METHOD PRIVATE T13_TestPowerForTopElement
VAR_INST
	iStep: INT;
END_VAR
IF (TcUnit.TEST_ORDERED ('T13_TestPowerForTopElement')) THEN
	GVL_Variable.fbPB1.ExecuteEveryCycle_Test ();
	GVL_Variable.fbPB1.ExecuteEveryCycle_Operation ();
	GVL_Variable.fbPB1.ExecuteEveryCycle_Status ();
	 CASE iStep	OF
	0	:
		GVL.fbSS1.SetFlag (bState	:= FALSE);
		GVL.fbSTO.SetFlag (bState	:= FALSE);
		AssertFalse		(Condition := GVL.fbSS1.GetFlag (), Message := 'K0 - T01 - bledny stan SS1');
		AssertFalse		(Condition := GVL.fbSTO.GetFlag (), Message := 'K0 - T02 - bledny stan SSO');
		GVL_Variable.fbPB1.PowerTurnOn ();
		iStep			:= iStep + 10;
	10	:
		AssertFalse (Condition := GVL_Variable.fbPB1.stEvents.arrState [1], 				Message := 'T10 - 01 - bledny stan bledu SS1');
		AssertFalse (Condition := GVL_Variable.fbPB1.stEvents.arrState [2], 				Message := 'T10 - 02 - bledny stan bledu STO');
		AssertTrue (Condition := GVL_Variable.fbPB1.stPower.cmdTurnOn.IsBusy (), 			Message := 'T10 - 03 - bledny stan trwa');
		AssertTrue (Condition := GVL_Variable.fbPB1.stPower.cmdTurnOn.IsFirstCycle (), 	Message := 'T10 - 05 - bledny pierwszy cykl');
		AssertFalse (Condition := GVL_Variable.fbPB1.stPower.cmdTurnOn.IsLastCycle (), 	Message := 'T10 - 06 - bledny ostatni cykl');
		AssertFalse (Condition := GVL_Variable.fbPB1.PowerGetStatus (), 					Message := 'T10 - 04 - bledny status');
		iStep			:= iStep + 10;
	20	:
		AssertTrue (Condition := GVL_Variable.fbPB1.stEvents.arrState [1], 					Message := 'T20 - 01 - bledny stan bledu SS1');
		AssertTrue (Condition := GVL_Variable.fbPB1.stEvents.arrState [2], 					Message := 'T20 - 02 - bledny stan bledu STO');
		AssertFalse (Condition := GVL_Variable.fbPB1.stPower.cmdTurnOn.IsBusy (), 			Message := 'T20 - 03 - bledny stan trwa');
		AssertFalse (Condition := GVL_Variable.fbPB1.stPower.cmdTurnOn.IsFirstCycle (),	Message := 'T20 - 05 - bledny pierwszy cykl');
		AssertFalse (Condition := GVL_Variable.fbPB1.stPower.cmdTurnOn.IsLastCycle (),	 	Message := 'T20 - 06 - bledny ostatni cykl');
		AssertFalse (Condition := GVL_Variable.fbPB1.PowerGetStatus (), 					Message := 'T20 - 04 - bledny status');
		GVL.fbSS1.SetFlag (bState	:= TRUE);
		GVL.fbSTO.SetFlag (bState	:= TRUE);
		iStep			:= iStep + 10;
	30	:
		iStep			:= iStep + 10;
	40	:
		GVL_Variable.fbPB1.PowerTurnOn ();
		iStep 			:= iStep + 10;
	50	:
		AssertTrue (Condition := GVL_Variable.fbPB1.stEvents.arrState [1], 				Message := 'T50 - 01 - bledny stan bledu SS1');
		AssertTrue (Condition := GVL_Variable.fbPB1.stEvents.arrState [2], 				Message := 'T50 - 02 - bledny stan bledu STO');
		AssertTrue (Condition := GVL_Variable.fbPB1.stPower.cmdTurnOn.IsBusy (), 		Message := 'T50 - 03 - bledny stan trwa');
		AssertFalse (Condition := GVL_Variable.fbPB1.PowerGetStatus (), 					Message := 'T50 - 04 - bledny status');
		iStep			:= iStep + 10;
	60	:
		AssertFalse (Condition := GVL_Variable.fbPB1.stEvents.arrState [1], 			Message := 'T60 - 01 - bledny stan bledu SS1');
		AssertFalse (Condition := GVL_Variable.fbPB1.stEvents.arrState [2], 			Message := 'T60 - 02 - bledny stan bledu STO');
		AssertTrue (Condition := GVL_Variable.fbPB1.stPower.cmdTurnOn.IsBusy (), 		Message := 'T60 - 03 - bledny stan trwa');
		AssertFalse (Condition := GVL_Variable.fbPB1.PowerGetStatus (), 					Message := 'T60 - 04 - bledny status');
		iStep			:= iStep + 10;
	70	:
		AssertTrue (Condition := GVL_Variable.fbPB1.stPower.cmdTurnOn.IsBusy (), 		Message := 'T70 - 03 - bledny stan trwa');
		AssertFalse (Condition := GVL_Variable.fbPB1.PowerGetStatus (), 					Message := 'T70 - 04 - bledny status');
		iStep			:= iStep + 10;
	80	:
		AssertTrue (Condition := GVL_Variable.fbPB1.stPower.cmdTurnOn.IsBusy (), 		Message := 'T80 - 03 - bledny stan trwa');
		AssertFalse (Condition := GVL_Variable.fbPB1.PowerGetStatus (), 					Message := 'T80 - 04 - bledny status');
		iStep			:= iStep + 10;
	90	:
		AssertTrue (Condition := GVL_Variable.fbPB1.stPower.cmdTurnOn.IsBusy (), 		Message := 'T90 - 03 - bledny stan trwa');
		AssertFalse (Condition := GVL_Variable.fbPB1.PowerGetStatus (), 					Message := 'T90 - 04 - bledny status');
		iStep			:= iStep + 10;
	100	:
		AssertTrue (Condition := GVL_Variable.fbPB1.stPower.cmdTurnOn.IsBusy (), 		Message := 'T100 - 03 - bledny stan trwa');
		AssertFalse (Condition := GVL_Variable.fbPB1.PowerGetStatus (), 					Message := 'T100 - 04 - bledny status');
		iStep			:= iStep + 10;
	110	:
		AssertTrue (Condition := GVL_Variable.fbPB1.stPower.cmdTurnOn.IsBusy (), 		Message := 'T110 - 03 - bledny stan trwa');
		AssertFalse (Condition := GVL_Variable.fbPB1.PowerGetStatus (), 					Message := 'T110 - 04 - bledny status');
		iStep			:= iStep + 10;
	120	:
		AssertTrue (Condition := GVL_Variable.fbPB1.stPower.cmdTurnOn.IsBusy (), 		Message := 'T120 - 03 - bledny stan trwa');
		AssertTrue (Condition := GVL_Variable.fbPB1.PowerGetStatus (), 					Message := 'T120 - 04 - bledny status');
		iStep			:= iStep + 10;
	130	:
		AssertFalse (Condition := GVL_Variable.fbPB1.stPower.cmdTurnOn.IsBusy (), 	Message := 'T130 - 03 - bledny stan trwa');
		AssertTrue (Condition := GVL_Variable.fbPB1.PowerGetStatus (), 					Message := 'T130 - 04 - bledny status');
		iStep			:= iStep + 10;
	140	:
		iStep			:= iStep + 10;
	150	:
		GVL_Variable.fbPB1.PowerTurnOff ();
		iStep			:= iStep + 10;
	160	:
		AssertTrue (Condition := GVL_Variable.fbPB1.stPower.cmdTurnOff.IsBusy (), 	Message := 'T160 - 03 - bledny stan trwa');
		AssertTrue (Condition := GVL_Variable.fbPB1.PowerGetStatus (), 					Message := 'T160 - 04 - bledny status');
		iStep			:= iStep + 10;
	170	:
		AssertTrue (Condition := GVL_Variable.fbPB1.stPower.cmdTurnOff.IsBusy (), 	Message := 'T170 - 03 - bledny stan trwa');
		AssertTrue (Condition := GVL_Variable.fbPB1.PowerGetStatus (), 					Message := 'T170 - 04 - bledny status');
		iStep			:= iStep + 10;
	180	:
		AssertTrue (Condition := GVL_Variable.fbPB1.stPower.cmdTurnOff.IsBusy (), 	Message := 'T180 - 03 - bledny stan trwa');
		AssertTrue (Condition := GVL_Variable.fbPB1.PowerGetStatus (), 					Message := 'T180 - 04 - bledny status');
		iStep			:= iStep + 10;
	190	:
		AssertTrue (Condition := GVL_Variable.fbPB1.stPower.cmdTurnOff.IsBusy (), 	Message := 'T190 - 03 - bledny stan trwa');
		AssertTrue (Condition := GVL_Variable.fbPB1.PowerGetStatus (), 					Message := 'T190 - 04 - bledny status');
		iStep			:= iStep + 10;
	200	:
		AssertTrue (Condition := GVL_Variable.fbPB1.stPower.cmdTurnOff.IsBusy (), 	Message := 'T200 - 03 - bledny stan trwa');
		AssertTrue (Condition := GVL_Variable.fbPB1.PowerGetStatus (), 					Message := 'T200 - 04 - bledny status');
		iStep			:= iStep + 10;
	210	:
		AssertTrue (Condition := GVL_Variable.fbPB1.stPower.cmdTurnOff.IsBusy (), 	Message := 'T210 - 03 - bledny stan trwa');
		AssertTrue (Condition := GVL_Variable.fbPB1.PowerGetStatus (), 					Message := 'T210 - 04 - bledny status');
		iStep			:= iStep + 10;
	220	:
		AssertTrue (Condition := GVL_Variable.fbPB1.stPower.cmdTurnOff.IsBusy (), 	Message := 'T220 - 03 - bledny stan trwa');
		AssertTrue (Condition := GVL_Variable.fbPB1.PowerGetStatus (), 					Message := 'T220 - 04 - bledny status');
		iStep			:= iStep + 10;
	230	:
		AssertTrue (Condition := GVL_Variable.fbPB1.stPower.cmdTurnOff.IsBusy (), 	Message := 'T230 - 03 - bledny stan trwa');
		AssertFalse (Condition := GVL_Variable.fbPB1.PowerGetStatus (), 					Message := 'T230 - 04 - bledny status');
		iStep		:= 1000;
	1000	:
		TcUnit.TEST_FINISHED ();
	END_CASE
END_IF
END_METHOD

METHOD PRIVATE T14_TestHomingControlElementWithouutHomingMethod
VAR_INST
	iStep			: INT;
END_VAR
IF (TcUnit.TEST_ORDERED ('T14_TestHomingControlElementWithouutHomingMethod')) THEN

	GVL_Variable.fbPB1_Wyk1.ExecuteEveryCycle_Test ();
	GVL_Variable.fbPB1_Wyk1.ExecuteEveryCycle_Operation ();
	GVL_Variable.fbPB1_Wyk1.ExecuteEveryCycle_Status ();
	GVL_Variable.fbPB1_Wyk1.ExecuteEveryCycle_Error ();

	CASE iStep OF
	0	:	
		GVL_Variable.fbPB1_Wyk1.PowerTurnOn ();
		iStep		:= iStep + 10;
	10	:
		IF (GVL_Variable.fbPB1_Wyk1.PowerGetStatus ()) THEN
			iStep	:= iStep + 10;
		END_IF
	20	:
		GVL_Variable.fbPB1_Wyk1.HomingStart ();
		iStep		:= iStep + 10;
	30	:
		//start cyklu
		AssertTrue (Condition := GVL_Variable.fbPB1_Wyk1.HomingGetBusy (), 		Message := 'S30 - T01 - Blad trwa');
		AssertFalse (Condition := GVL_Variable.fbPB1_Wyk1.HomingGetDone (), 	Message := 'S30 - T02 - Blad gotowe');
		AssertTrue (Condition := GVL_Variable.fbPB1_Wyk1.HomingGetIsNeeded (), 	Message := 'S30 - T02 - Blad potrzebne');
		iStep		:= iStep + 10;
	40	:	
		//trwa\
		AssertTrue (Condition := GVL_Variable.fbPB1_Wyk1.HomingGetBusy (), 		Message := 'S40 - T01 -Blad trwa');     
		AssertFalse (Condition := GVL_Variable.fbPB1_Wyk1.HomingGetDone (),		Message := 'S40 - T02 -Blad gotowe');   
		AssertTrue (Condition := GVL_Variable.fbPB1_Wyk1.HomingGetIsNeeded (), 	Message := 'S40 - T02 -Blad potrzebne');
		iStep		:= iStep + 10;
	50	:
		//trwa\
		AssertTrue (Condition := GVL_Variable.fbPB1_Wyk1.HomingGetBusy (), 		Message := 'S50 - T01 - Blad trwa');     
		AssertFalse (Condition := GVL_Variable.fbPB1_Wyk1.HomingGetDone (),		Message := 'S50 - T02 - Blad gotowe');   
		AssertTrue (Condition := GVL_Variable.fbPB1_Wyk1.HomingGetIsNeeded (), 	Message := 'S50 - T02 - Blad potrzebne');
		iStep		:= iStep + 10;
	60	:
		//koniec cyklu
		AssertTrue (Condition := GVL_Variable.fbPB1_Wyk1.HomingGetBusy (),		Message := 'S60 - T01 - Blad trwa');     
		AssertFalse (Condition := GVL_Variable.fbPB1_Wyk1.HomingGetDone (), 	Message := 'S60 - T02 - Blad gotowe');   
		AssertFalse (Condition := GVL_Variable.fbPB1_Wyk1.HomingGetIsNeeded (), Message := 'S60 - T02 - Blad potrzebne');
		iStep		:= iStep + 10;
	70	:
		//last cycle
		AssertFalse (Condition := GVL_Variable.fbPB1_Wyk1.HomingGetBusy (),		Message := 'S70 - T01 - Blad trwa');     
		AssertTrue (Condition := GVL_Variable.fbPB1_Wyk1.HomingGetDone (), 		Message := 'S70 - T02 - Blad gotowe');   
		AssertFalse (Condition := GVL_Variable.fbPB1_Wyk1.HomingGetIsNeeded (), Message := 'S70 - T02 - Blad potrzebne');
	
		iStep		:= 1000;
	1000	:
		TcUnit.TEST_FINISHED ();
	END_CASE
END_IF
END_METHOD

METHOD PRIVATE T15_TestHomingControlElementWithHomingMetod
VAR_INST
	iStep			: INT;
END_VAR
IF (TcUnit.TEST_ORDERED ('T15_TestHomingControlElementWithHomingMetod')) THEN

	GVL_Variable.fbPB1_Wyk2.ExecuteEveryCycle_Test ();
	GVL_Variable.fbPB1_Wyk2.ExecuteEveryCycle_Operation ();
	GVL_Variable.fbPB1_Wyk2.ExecuteEveryCycle_Status ();
	GVL_Variable.fbPB1_Wyk2.ExecuteEveryCycle_Error ();

	CASE iStep OF
	0	:	
		GVL_Variable.fbPB1_Wyk2.PowerTurnOn ();
		iStep		:= iStep + 10;
	10	:
		IF (GVL_Variable.fbPB1_Wyk2.PowerGetStatus ()) THEN
			iStep	:= iStep + 10;
		END_IF
	20	:
		GVL_Variable.fbPB1_Wyk2.HomingStart ();
		iStep		:= iStep + 10;
	30	:
		//start cyklu
		AssertTrue (Condition := GVL_Variable.fbPB1_Wyk2.HomingGetBusy (), 		Message := 'S30 - T01 - Blad trwa');
		AssertFalse (Condition := GVL_Variable.fbPB1_Wyk2.HomingGetDone (), 	Message := 'S30 - T02 - Blad gotowe');
		AssertTrue (Condition := GVL_Variable.fbPB1_Wyk2.HomingGetIsNeeded (), 	Message := 'S30 - T02 - Blad potrzebne');
		iStep		:= iStep + 10;
	40	:	
		//trwa\
		AssertTrue (Condition := GVL_Variable.fbPB1_Wyk2.HomingGetBusy (), 		Message := 'S40 - T01 -Blad trwa');     
		AssertFalse (Condition := GVL_Variable.fbPB1_Wyk2.HomingGetDone (),		Message := 'S40 - T02 -Blad gotowe');   
		AssertTrue (Condition := GVL_Variable.fbPB1_Wyk2.HomingGetIsNeeded (), 	Message := 'S40 - T02 -Blad potrzebne');
		iStep		:= iStep + 10;
	50	:
		//trwa\
		AssertTrue (Condition := GVL_Variable.fbPB1_Wyk2.HomingGetBusy (), 		Message := 'S50 - T01 - Blad trwa');     
		AssertFalse (Condition := GVL_Variable.fbPB1_Wyk2.HomingGetDone (),		Message := 'S50 - T02 - Blad gotowe');   
		AssertTrue (Condition := GVL_Variable.fbPB1_Wyk2.HomingGetIsNeeded (), 	Message := 'S50 - T02 - Blad potrzebne');
		iStep		:= iStep + 10;
	60	: 
		WRITE_PROTECTED_BOOL (Ptr := ADR (GVL_Variable.fbPB1_Wyk2.bHomingFinished), Value := TRUE);
		iStep		:= iStep + 10;
	70	:	
		//trwa\
		AssertTrue (Condition := GVL_Variable.fbPB1_Wyk2.HomingGetBusy (), 		Message := 'S70 - T01 -Blad trwa');     
		AssertFalse (Condition := GVL_Variable.fbPB1_Wyk2.HomingGetDone (),		Message := 'S70 - T02 -Blad gotowe');   
		AssertTrue (Condition := GVL_Variable.fbPB1_Wyk2.HomingGetIsNeeded (), 	Message := 'S70 - T02 -Blad potrzebne');
		iStep		:= iStep + 10;
	80	:
		//trwa\
		AssertTrue (Condition := GVL_Variable.fbPB1_Wyk2.HomingGetBusy (), 		Message := 'S80 - T01 - Blad trwa');     
		AssertFalse (Condition := GVL_Variable.fbPB1_Wyk2.HomingGetDone (),		Message := 'S80 - T02 - Blad gotowe');   
		AssertTrue (Condition := GVL_Variable.fbPB1_Wyk2.HomingGetIsNeeded (), 	Message := 'S80 - T02 - Blad potrzebne');
		iStep		:= iStep + 10;
		
		
		
	90	:
		//koniec cyklu
		AssertTrue (Condition := GVL_Variable.fbPB1_Wyk2.HomingGetBusy (),		Message := 'S90 - T01 - Blad trwa');     
		AssertFalse (Condition := GVL_Variable.fbPB1_Wyk2.HomingGetDone (), 	Message := 'S90 - T02 - Blad gotowe');   
		AssertFalse (Condition := GVL_Variable.fbPB1_Wyk2.HomingGetIsNeeded (), Message := 'S90 - T02 - Blad potrzebne');
		iStep		:= iStep + 10;
	100	:
		//last cycle
		AssertFalse (Condition := GVL_Variable.fbPB1_Wyk2.HomingGetBusy (),		Message := 'S100 - T01 - Blad trwa');     
		AssertTrue (Condition := GVL_Variable.fbPB1_Wyk2.HomingGetDone (), 		Message := 'S100 - T02 - Blad gotowe');   
		AssertFalse (Condition := GVL_Variable.fbPB1_Wyk2.HomingGetIsNeeded (), Message := 'S100 - T02 - Blad potrzebne');
	
		iStep		:= 1000;
	1000	:
		TcUnit.TEST_FINISHED ();
	END_CASE
END_IF
END_METHOD

METHOD PRIVATE T16_TestingTopElementHoming
VAR_INST
	iStep	: INT;
END_VAR
IF (TcUnit.TEST_ORDERED ('T16_TestingTopElementHoming')) THEN

	GVL_Variable.fbPB1.ExecuteEveryCycle_Test ();
	GVL_Variable.fbPB1.ExecuteEveryCycle_Operation ();
	GVL_Variable.fbPB1.ExecuteEveryCycle_Status ();
	GVL_Variable.fbPB1.ExecuteEveryCycle_Error ();

	CASE iStep OF
	0	:
		GVL_Variable.fbPB1.PowerTurnOn ();
		iStep		:= iStep + 10;
	10	:
		IF (GVL_Variable.fbPB1.PowerGetStatus ()) THEN
			iStep	:= iStep + 10;
		END_IF
	20	:
		GVL_Variable.fbPB1.HomingStart ();
		iStep		:= iStep + 10;
	30	:
		AssertTrue (Condition := GVL_Variable.fbPB1.HomingGetBusy (), 			Message := 'S30 - T01');
		AssertFalse (Condition := GVL_Variable.fbPB1_Wyk1.HomingGetBusy (),		Message := 'S30 - T02');
		AssertFalse (Condition := GVL_Variable.fbPB1_Wyk2.HomingGetBusy (),		Message := 'S30 - T03');
		AssertFalse (Condition := GVL_Variable.fbPB1_ZL1.HomingGetBusy (), 		Message := 'S30 - T04');
		AssertFalse (Condition := GVL_Variable.fbPB1_ZL1_Wyk1.HomingGetBusy (),	Message := 'S30 - T05');
		AssertFalse (Condition := GVL_Variable.fbPB1_ZL1_Wyk2.HomingGetBusy (),	Message := 'S30 - T06');

		AssertFalse (Condition := GVL_Variable.fbPB1.HomingGetDone (), 			Message := 'S30 - T07');
		AssertTrue (Condition := GVL_Variable.fbPB1_Wyk1.HomingGetDone (),		Message := 'S30 - T08');
		AssertTrue (Condition := GVL_Variable.fbPB1_Wyk2.HomingGetDone (),		Message := 'S30 - T09');
		AssertFalse (Condition := GVL_Variable.fbPB1_ZL1.HomingGetDone (), 		Message := 'S30 - T10');
		AssertFalse (Condition := GVL_Variable.fbPB1_ZL1_Wyk1.HomingGetDone (),	Message := 'S30 - T11');
		AssertFalse (Condition := GVL_Variable.fbPB1_ZL1_Wyk2.HomingGetDone (),	Message := 'S30 - T12');
		iStep		:= iStep + 10;
	40	:
		AssertTrue (Condition := GVL_Variable.fbPB1.HomingGetBusy (), 			Message := 'S40 - T01');
		AssertTrue (Condition := GVL_Variable.fbPB1_Wyk1.HomingGetBusy (),		Message := 'S40 - T02');
		AssertTrue (Condition := GVL_Variable.fbPB1_Wyk2.HomingGetBusy (),		Message := 'S40 - T03');
		AssertTrue (Condition := GVL_Variable.fbPB1_ZL1.HomingGetBusy (), 		Message := 'S40 - T04');
		AssertTrue (Condition := GVL_Variable.fbPB1_ZL1_Wyk1.HomingGetBusy (),	Message := 'S40 - T05');
		AssertTrue (Condition := GVL_Variable.fbPB1_ZL1_Wyk2.HomingGetBusy (),	Message := 'S40 - T06');

		AssertFalse (Condition := GVL_Variable.fbPB1.HomingGetDone (), 			Message := 'S40 - T07');
		AssertFalse (Condition := GVL_Variable.fbPB1_Wyk1.HomingGetDone (),		Message := 'S40 - T08');
		AssertFalse (Condition := GVL_Variable.fbPB1_Wyk2.HomingGetDone (),		Message := 'S40 - T09');
		AssertFalse (Condition := GVL_Variable.fbPB1_ZL1.HomingGetDone (), 		Message := 'S40 - T10');
		AssertFalse (Condition := GVL_Variable.fbPB1_ZL1_Wyk1.HomingGetDone (),	Message := 'S40 - T11');
		AssertFalse (Condition := GVL_Variable.fbPB1_ZL1_Wyk2.HomingGetDone (),	Message := 'S40 - T12');
		iStep		:= iStep + 10;
	50	:
		AssertTrue (Condition := GVL_Variable.fbPB1.HomingGetBusy (), 			Message := 'S50 - T01');
		AssertTrue (Condition := GVL_Variable.fbPB1_Wyk1.HomingGetBusy (),		Message := 'S50 - T02');
		AssertTrue (Condition := GVL_Variable.fbPB1_Wyk2.HomingGetBusy (),		Message := 'S50 - T03');
		AssertTrue (Condition := GVL_Variable.fbPB1_ZL1.HomingGetBusy (), 		Message := 'S50 - T04');
		AssertTrue (Condition := GVL_Variable.fbPB1_ZL1_Wyk1.HomingGetBusy (),	Message := 'S50 - T05');
		AssertTrue (Condition := GVL_Variable.fbPB1_ZL1_Wyk2.HomingGetBusy (),	Message := 'S50 - T06');

		AssertFalse (Condition := GVL_Variable.fbPB1.HomingGetDone (), 			Message := 'S50 - T07');
		AssertFalse (Condition := GVL_Variable.fbPB1_Wyk1.HomingGetDone (),		Message := 'S50 - T08');
		AssertFalse (Condition := GVL_Variable.fbPB1_Wyk2.HomingGetDone (),		Message := 'S50 - T09');
		AssertFalse (Condition := GVL_Variable.fbPB1_ZL1.HomingGetDone (), 		Message := 'S50 - T10');
		AssertFalse (Condition := GVL_Variable.fbPB1_ZL1_Wyk1.HomingGetDone (),	Message := 'S50 - T11');
		AssertFalse (Condition := GVL_Variable.fbPB1_ZL1_Wyk2.HomingGetDone (),	Message := 'S50 - T12');
		iStep		:= iStep + 10;
		
		
		iStep		:= 1000;
	1000	:
		TcUnit.TEST_FINISHED ();
	END_CASE
END_IF
END_METHOD

METHOD PROTECTED T20_TestCommunicator
VAR
	bResult		: BOOL;
	bWartosc	: BOOL;
	itfSender		: ITF_BaseMessengerSender;
	itfRecipient	: ITF_BaseMessengerRecipient;
	itftmpSender	: ITF_BaseMessengerSender;
	itftmpRecipient	: ITF_BaseMessengerRecipient;
END_VAR
IF (TcUnit.TEST_ORDERED ('T20_TestCommunicator')) THEN
	GVL_Variable.fbClientComm1.LinkCommunicator (fbCommunicator := GVL.fbCommunicator);
	GVL_Variable.fbClientComm2.LinkCommunicator (fbCommunicator := GVL.fbCommunicator);
	GVL_Variable.fbClientComm3.LinkCommunicator (fbCommunicator := GVL.fbCommunicator);
	GVL_Variable.fbClientComm4.LinkCommunicator (fbCommunicator := GVL.fbCommunicator);
	GVL_Variable.fbClientComm5.LinkCommunicator (fbCommunicator := GVL.fbCommunicator);
	GVL_Variable.fbClientComm6.LinkCommunicator (fbCommunicator := GVL.fbCommunicator);
	
	GVL.fbCommunicator.AddMessage (sText := 'Test1');
	AssertEquals_INT (Expected := 1, Actual := GVL.fbCommunicator.iNumberOfData, Message := 'T01a- bledna ilosc komunikatow');
	GVL.fbCommunicator.AddMessage (sText := 'Test2');
	AssertEquals_INT (Expected := 2, Actual := GVL.fbCommunicator.iNumberOfData, Message := 'T01b- bledna ilosc komunikatow');
	GVL.fbCommunicator.AddMessage (sText := 'Test3');
	AssertEquals_INT (Expected := 3, Actual := GVL.fbCommunicator.iNumberOfData, Message := 'T01c- bledna ilosc komunikatow');
//dodawanie klientów
	GVL.fbCommunicator.AddSenderToMessage (iMessageNumber := 1, itfSender := GVL_Variable.fbClientComm1);
	itfSender			:= GVL_Variable.fbClientComm1;
	itftmpSender		:= GVL.fbCommunicator.arrData [1].itfSender;
	
	AssertEquals (Expected := itfSender, Actual := itftmpSender, Message := 'T01 - bledny nadawca');
	
	GVL.fbCommunicator.AddSenderToMessage (iMessageNumber := 2, itfSender := GVL_Variable.fbClientComm2);
	itfSender			:= GVL_Variable.fbClientComm2;
	itftmpSender		:= GVL.fbCommunicator.arrData [2].itfSender;
	AssertEquals (Expected := itfSender, Actual := itftmpSender, Message := 'T02 - bledny nadawca');

	GVL.fbCommunicator.AddSenderToMessage (iMessageNumber := 3, itfSender := GVL_Variable.fbClientComm3);
	itfSender			:= GVL_Variable.fbClientComm3;
	itftmpSender		:= GVL.fbCommunicator.arrData [3].itfSender;
	AssertEquals (Expected := itfSender, Actual := itftmpSender, Message := 'T03 - bledny nadawca');

//Przypisanie odbiorców

	GVL.fbCommunicator.AddRecipientToMessage (iMessageNumber := 1, itfRecipient := GVL_Variable.fbClientComm4);
	itfRecipient		:= GVL_Variable.fbClientComm4;
	itftmpRecipient		:= GVL.fbCommunicator.arrData [1].arritfRecipient [1];
	AssertEquals (Expected := itfRecipient, Actual := itftmpRecipient, Message := 'T04 - bledny odbiorca');
//	
	GVL.fbCommunicator.AddRecipientToMessage (iMessageNumber := 2, itfRecipient := GVL_Variable.fbClientComm1);
	itfRecipient		:= GVL_Variable.fbClientComm1;
	itftmpRecipient		:= GVL.fbCommunicator.arrData [2].arritfRecipient [1];
	AssertEquals (Expected := itfRecipient, Actual := itftmpRecipient, Message := 'T05 - bledny odbiorca');
	
	GVL.fbCommunicator.AddRecipientToMessage (iMessageNumber := 2, itfRecipient := GVL_Variable.fbClientComm5);
	itfRecipient		:= GVL_Variable.fbClientComm5;
	itftmpRecipient		:= GVL.fbCommunicator.arrData [2].arritfRecipient [2];
	AssertEquals (Expected := itfRecipient, Actual := itftmpRecipient, Message := 'T05b - bledny odbiorca');
	
	GVL.fbCommunicator.AddRecipientToMessage (iMessageNumber := 2, itfRecipient := GVL_Variable.fbClientComm6);
	itfRecipient		:= GVL_Variable.fbClientComm6;
	itftmpRecipient		:= GVL.fbCommunicator.arrData [2].arritfRecipient [3];
	AssertEquals (Expected := itfRecipient, Actual := itftmpRecipient, Message := 'T05c - bledny odbiorca');
//	
	GVL.fbCommunicator.AddRecipientToMessage (iMessageNumber := 3, itfRecipient := GVL_Variable.fbClientComm5);
	itfRecipient		:= GVL_Variable.fbClientComm5;
	itftmpRecipient		:= GVL.fbCommunicator.arrData [3].arritfRecipient [1];
	AssertEquals (Expected := itfRecipient, Actual := itftmpRecipient, Message := 'T06 - bledny odbiorca');

//Test nadawanie
	bResult := GVL_Variable.fbClientComm1.Send_BOOL (sText := 'Test1');
	AssertTrue (Condition := bResult, 														Message := 'T02a - Blad nadania');
	AssertEquals_INT (Expected := 1, Actual := GVL.fbCommunicator.iNumberOfitemsInStack, 	Message := 'T02b - bledna dlugosc kolejki');
	AssertTrue (Condition := GVL.fbCommunicator.arrStack [1].stMessage.bValue, 				Message := 'T02c - baledna wartosc w kolejce');
	AssertEquals_STRING (Expected := 'Test1', Actual := GVL.fbCommunicator.arrStack [1].stMessage.sText, Message := 'T02d - Bladna nazwa komunikatu');
	
	GVL.fbCommunicator.StackSupport ();
	AssertEquals_INT (Expected := 0, Actual := GVL.fbCommunicator.iNumberOfitemsInStack, 	Message := 'T04a - bledna dlugosc kolejki');
	AssertFalse (Condition := GVL.fbCommunicator.arrStack [1].stMessage.bValue, 				Message := 'T04b - Bledna wartosc');
	
	bResult	:= GVL_Variable.fbClientComm1.Receive_BOOL (sText := 'Test1', bValue => bWartosc);
	AssertFalse	(Condition := bResult, 														Message := 'T04c - blaedna zgoda na odczyt wiadomosci');
	AssertFalse (Condition := bWartosc, 													Message := 'T04d - blednie odczytana wartosc');

	bResult	:= GVL_Variable.fbClientComm4.Receive_BOOL (sText := 'Test1', bValue => bWartosc);
	AssertTrue	(Condition := bResult, 														Message := 'T04e - blaedna zgoda na odczyt wiadomosci');
	AssertTrue (Condition := bWartosc, 														Message := 'T04f - blednie odczytana wartosc');
	
	bResult	:= GVL_Variable.fbClientComm1.ConfirmReceipt (sText := 'Test1');
	Assertfalse	(Condition := bResult, 														Message := 'T04g - powierdzone choc nie mozna');

	AssertEquals_INT (Expected := 0, Actual := GVL.fbCommunicator.iNumberOfitemsInStack, 	Message := 'T04h - bledna dlugosc kolejki');
	GVL.fbCommunicator.StackSupport ();
	AssertEquals_INT (Expected := 0, Actual := GVL.fbCommunicator.iNumberOfitemsInStack, 	Message := 'T04i - bledna dlugosc kolejki');
	AssertFalse (Condition := GVL.fbCommunicator.arrStack [1].stMessage.bValue, 			Message := 'T04j - Bledna wartosc');
	
	bResult	:= GVL_Variable.fbClientComm4.ConfirmReceipt (sText := 'Test1');
	AssertTrue	(Condition := bResult, 														Message := 'T04k - nie powierdzone choc mozna');

	AssertEquals_INT (Expected := 1, Actual := GVL.fbCommunicator.iNumberOfitemsInStack, 	Message := 'T04l - bledna dlugosc kolejki');
	GVL.fbCommunicator.StackSupport ();
	AssertEquals_INT (Expected := 0, Actual := GVL.fbCommunicator.iNumberOfitemsInStack, 	Message := 'T04m - bledna dlugosc kolejki');
	Assertfalse (Condition := GVL.fbCommunicator.arrStack [1].stMessage.bValue, 			Message := 'T04n - Bledna wartosc');	
//Nadawanie do kilku odbiorców
//Nadanie komunikatu
	bResult	:= GVL_Variable.fbClientComm2.Send_BOOL (sText := 'Test2');
	AssertTrue (Condition := bResult, 														Message := 'T05a - Blad nadania');
	AssertEquals_STRING (Expected := 'Test2', Actual := GVL.fbCommunicator.arrStack [1].stMessage.sText, 	Message := 'T05b - Bladna nazwa komunikatu');
	AssertTrue (Condition := GVL.fbCommunicator.arrStack [1].stMessage.bValue,				Message := 'T05c - baledna wartosc w kolejce');
	
//Obsluga kolejki
	AssertEquals_INT (Expected := 1, Actual := GVL.fbCommunicator.iNumberOfitemsInStack, 	Message := 'T05d - bledna dlugosc kolejki');
	GVL.fbCommunicator.StackSupport ();
	AssertEquals_INT (Expected := 0, Actual := GVL.fbCommunicator.iNumberOfitemsInStack, 	Message := 'T05e - bledna dlugosc kolejki');
	AssertTrue (Condition := GVL.fbCommunicator.arrData [2].stMessage.bValue,				Message := 'T05f - Bledna wartosc');
	
//Odebranie  przez pierwszego klienta
	AssertEquals_INT (Expected := 3, Actual := GVL.fbCommunicator.arrData [2].iNumberOfConfirmations,	Message := 'T05g - bledna ilosc odbiorcow krzorzy maja potwierdzic');
	bResult	:= GVL_Variable.fbClientComm1.Receive_BOOL (sText := 'Test2', bValue => bWartosc);
	AssertTrue (Condition := bResult, 																	Message := 'T05h - Blad odbierania');
	AssertTrue (Condition := bWartosc,																	Message := 'T05i - bledna zmienna odebrana');

//Obsluga kolejki
	AssertEquals_INT (Expected := 0, Actual := GVL.fbCommunicator.iNumberOfitemsInStack, 				Message := 'T05j - bledna dlugosc kolejki');
	GVL.fbCommunicator.StackSupport ();
	AssertEquals_INT (Expected := 0, Actual := GVL.fbCommunicator.iNumberOfitemsInStack, 				Message := 'T05k - bledna dlugosc kolejki');
	AssertTrue (Condition := GVL.fbCommunicator.arrData [2].stMessage.bValue, 							Message := 'T05l - Bledna wartosc');
	
//potwierdzenie  przez pierwszego klienta
	AssertEquals_INT (Expected := 3, Actual := GVL.fbCommunicator.arrData [2].iNumberOfConfirmations,	Message := 'T05m - bledna ilosc odbiorcow krzorzy maja potwierdzic');
	bResult	:= GVL_Variable.fbClientComm1.ConfirmReceipt (sText := 'Test2');
	AssertTrue (Condition := bResult, 																	Message := 'T05n - Blad potwierdzenia');
	
//Obsluga kolejki
	AssertEquals_INT (Expected := 1, Actual := GVL.fbCommunicator.iNumberOfitemsInStack, 				Message := 'T05o - bledna dlugosc kolejki');
	GVL.fbCommunicator.StackSupport ();
	AssertEquals_INT (Expected := 0, Actual := GVL.fbCommunicator.iNumberOfitemsInStack, 				Message := 'T05p - bledna dlugosc kolejki');
	AssertTrue (Condition := GVL.fbCommunicator.arrData [2].stMessage.bValue, 							Message := 'T05r - Bledna wartosc');

(*	*)
//odebranie przez kolejnego odbiorce
	AssertEquals_INT (Expected := 2, Actual := GVL.fbCommunicator.arrData [2].iNumberOfConfirmations,	Message := 'T05s - bledna ilosc odbiorcow krzorzy maja potwierdzic');
	bResult	:= GVL_Variable.fbClientComm5.Receive_BOOL (sText := 'Test2', bValue => bWartosc);
	AssertTrue (Condition := bResult, 																	Message := 'T05t - Blad odbierania');
	AssertTrue (Condition := bWartosc,																	Message := 'T05u - bledna zmienna odebrana');

//Obsluga kolejki
	AssertEquals_INT (Expected := 0, Actual := GVL.fbCommunicator.iNumberOfitemsInStack, 				Message := 'T05w - bledna dlugosc kolejki');
	GVL.fbCommunicator.StackSupport ();
	AssertEquals_INT (Expected := 0, Actual := GVL.fbCommunicator.iNumberOfitemsInStack, 				Message := 'T05x - bledna dlugosc kolejki');
	AssertTrue (Condition := GVL.fbCommunicator.arrData [2].stMessage.bValue, 							Message := 'T05y - Bledna wartosc');

//odebranie i potwierdszenie przez ostatniego odbiorce
	AssertEquals_INT (Expected := 2, Actual := GVL.fbCommunicator.arrData [2].iNumberOfConfirmations,	Message := 'T05z - bledna ilosc odbiorcow krzorzy maja potwierdzic');
	bResult	:= GVL_Variable.fbClientComm6.Receive_BOOL (sText := 'Test2', bValue => bWartosc);
	AssertTrue (Condition := bResult, 																	Message := 'T06a - Blad odbierania');
	AssertTrue (Condition := bWartosc,																	Message := 'T06b - bledna zmienna odebrana');

	bResult	:= GVL_Variable.fbClientComm6.ConfirmReceipt (sText := 'Test2');
	AssertTrue (Condition := bResult, 																	Message := 'T06c - Blad potwierdzania');

//Obsluga kolejki
	AssertEquals_INT (Expected := 1, Actual := GVL.fbCommunicator.iNumberOfitemsInStack, 				Message := 'T06d - bledna dlugosc kolejki');
	GVL.fbCommunicator.StackSupport ();
	AssertEquals_INT (Expected := 0, Actual := GVL.fbCommunicator.iNumberOfitemsInStack, 				Message := 'T06e - bledna dlugosc kolejki');
	AssertTrue (Condition := GVL.fbCommunicator.arrData [2].stMessage.bValue, 							Message := 'T06f - Bledna wartosc');

//potwierdzenie przez ostatniego
	bResult	:= GVL_Variable.fbClientComm5.ConfirmReceipt (sText := 'Test2');
	AssertTrue (Condition := bResult, 																	Message := 'T06g - Blad potwierdzania');

//Obsluga kolejki
	AssertEquals_INT (Expected := 1, Actual := GVL.fbCommunicator.iNumberOfitemsInStack, 				Message := 'T06h - bledna dlugosc kolejki');
	GVL.fbCommunicator.StackSupport ();
	AssertEquals_INT (Expected := 0, Actual := GVL.fbCommunicator.iNumberOfitemsInStack, 				Message := 'T06i - bledna dlugosc kolejki');
	AssertFalse (Condition := GVL.fbCommunicator.arrData [2].stMessage.bValue, 							Message := 'T06j - Bledna wartosc');

	AssertEquals_INT (Expected := 0, Actual := GVL.fbCommunicator.arrData [2].iNumberOfConfirmations,	Message := 'T06k - bledna ilosc odbiorcow do potwierdzenia');
	
	TcUnit.TEST_FINISHED ();
END_IF
END_METHOD

METHOD PROTECTED T21_TestCreateTepmplate
VAR
	bResult: BOOL;
	sttmpSkladnik: ST_BaseDescriptor;
END_VAR
IF (TcUnit.TEST_ORDERED ('T21_TestCreateTepmplate')) THEN
	//Dodanie zewnętreznego FB do twoerzenia szbalonów
	GVL.fbRecipe.AddITFToCreateTemplate (fbToCtreateTemplate := GVL.fbCreatingTemplate1);
	GVL.fbRecipe.AddITFToCreateTemplate (fbToCtreateTemplate := GVL.fbCreatingTemplate2);
	//wywołanie medody tworzacej szablony
	GVL.fbRecipe.CreateTemplates ();
	
	AssertEquals_UINT (Expected := 2, Actual := GVL.fbRecipe.GetNumberOfTemplate (), 'T01 - bledna ilosc szablonow');
	AssertEquals_UINT (Expected := 3, Actual := GVL.fbRecipe.GetNumberIngredientOFTemplate (uiNumber := 1), Message := 'T02 - bledna ilosc skladnikow');
	AssertEquals_UINT (Expected := 1, Actual := GVL.fbRecipe.GetNumberIngredientOFTemplate (uiNumber := 2), Message := 'T03 - bledna ilosc skladnikow');
	
	AssertEquals_WSTRING (Expected := "Nazwa skladnika 1 PL", Actual := GVL.fbRecipe.arrTemplates [1].arrIngredient [1].stTexts.arrText [1],	Message := 'Test 06b - bledna etykieta');
	AssertEquals_REAL (Expected := 1111, Actual := GVL.fbRecipe.arrTemplates [1].arrIngredient [1].rValue,										Message := 'Test 06c - bledna wartosc', Delta := 0);
	AssertEquals_REAL (Expected := 1111, Actual := GVL.fbRecipe.arrTemplates [1].arrIngredient [1].rDefaultValue,								Message := 'Test 06d - bledna wartosc domyslna', Delta := 0);
	AssertEquals_REAL (Expected := 1, Actual := GVL.fbRecipe.arrTemplates [1].arrIngredient [1].rMin,		 									Message := 'Test 06e - bledna wartosc min', Delta := 0);
	AssertEquals_REAL (Expected := 10000, Actual := GVL.fbRecipe.arrTemplates [1].arrIngredient [1].rMAX,		 								Message := 'Test 06f - bledna wartosc max', Delta := 0);
	AssertEquals_WSTRING (Expected := "mm", Actual := TO_WSTRING (GVL.fbRecipe.arrTemplates [1].arrIngredient [1].sUnit),		 				Message := 'Test 06g - bledna jednostka');
	
	AssertEquals_WSTRING (Expected := "Nazwa skladnika 2 PL", Actual := GVL.fbRecipe.arrTemplates [1].arrIngredient [2].stTexts.arrText [1],	Message := 'Test 07b - bledna etykieta');
	AssertEquals_REAL (Expected := 1112, Actual := GVL.fbRecipe.arrTemplates [1].arrIngredient [2].rValue,										Message := 'Test 07c - bledna wartosc', Delta := 0);
	AssertEquals_REAL (Expected := 1112, Actual := GVL.fbRecipe.arrTemplates [1].arrIngredient [2].rDefaultValue,								Message := 'Test 07d - bledna wartosc domyslna', Delta := 0);
	AssertEquals_REAL (Expected := 1, Actual := GVL.fbRecipe.arrTemplates [1].arrIngredient [2].rMin,		 									Message := 'Test 07e - bledna wartosc min', Delta := 0);
	AssertEquals_REAL (Expected := 10000, Actual := GVL.fbRecipe.arrTemplates [1].arrIngredient [2].rMAX,		 								Message := 'Test 07f - bledna wartosc max', Delta := 0);
	AssertEquals_WSTRING (Expected := "mm/s", Actual := TO_WSTRING (GVL.fbRecipe.arrTemplates [1].arrIngredient [2].sUnit),		 			Message := 'Test 07g - bledna jednostka');
	
//1 składnik 2 szablonu	
	AssertEquals_WSTRING (Expected := "Nazwa skladnika 1 PL", Actual := GVL.fbRecipe.arrTemplates [2].arrIngredient [1].stTexts.arrText [1],	Message := 'Test 11b - bledna etykieta');
	AssertEquals_REAL (Expected := 1111, Actual := GVL.fbRecipe.arrTemplates [2].arrIngredient [1].rValue,										Message := 'Test 11c - bledna wartosc', Delta := 0);
	AssertEquals_REAL (Expected := 1111, Actual := GVL.fbRecipe.arrTemplates [2].arrIngredient [1].rDefaultValue,								Message := 'Test 11d - bledna wartosc domyslna', Delta := 0);
	AssertEquals_REAL (Expected := 1, Actual := GVL.fbRecipe.arrTemplates [2].arrIngredient [1].rMin,		 									Message := 'Test 11e - bledna wartosc min', Delta := 0);
	AssertEquals_REAL (Expected := 10000, Actual := GVL.fbRecipe.arrTemplates [2].arrIngredient [1].rMAX,		 								Message := 'Test 11f - bledna wartosc max', Delta := 0);
	AssertEquals_WSTRING (Expected := "mm", Actual := TO_WSTRING (GVL.fbRecipe.arrTemplates [2].arrIngredient [1].sUnit),		 				Message := 'Test 11g - bledna jednostka');
	
	TcUnit.TEST_FINISHED ();
END_IF

(*
//Wyczyszczeni danych i test czyszczenia
	GVL.fbRecipe.DeleteRecipes ();
	GVL.fbRecipe.DeleteTemplates ();
	AssertEquals_UINT (Expected := 0, Actual := GVL.fbRecipe.GetNumberOfTemplate (), 			Message := 'T01 - bledna ilosc szablonow');
	AssertEquals_UINT (Expected := 0, Actual := GVL.fbRecipe.GetNumberOfRecipe (), 				Message := 'T02 - bledna ilosc receptur');
	AssertEquals_UINT (Expected := 0, Actual := GVL.fbRecipe.GetNumberOfChoosen (),	 			Message := 'T03 - bledny numer wybranej');
//	utworzenie szablonu z podaną nazwą
	GVL.fbRecipe.SetText (eLocation := E_BaseLocation.pl, wsDescription := "Nazwa szablonu PL");
	GVL.fbRecipe.SetText (eLocation := E_BaseLocation.en, wsDescription := "Nazwa szablonu EN");
	GVL.fbRecipe.SetText (eLocation := E_BaseLocation.de, wsDescription := "Nazwa szablonu DE");
	bResult	:= GVL.fbRecipe.AddTemplates (stTexts	:= GVL.fbRecipe.GetTexts ());
	AssertTrue (Condition := bResult,															Message := 'T04 - Blad utworzenia szablonu');
	AssertEquals_UINT (Expected := 1, Actual := GVL.fbRecipe.GetNumberOfTemplate (),			Message := 'T05 - Blad ilosci dodanych szablonow');
//dodawanie sładników
	GVL.fbRecipe.SetTextIn (stIN := sttmpSkladnik, eLocation := E_BaseLocation.pl, wsDescription := "Nazwa skladnika 1 PL");
	GVL.fbRecipe.SetTextIn (stIN := sttmpSkladnik, eLocation := E_BaseLocation.en, wsDescription := "Nazwa skladnika 1 EN");
	GVL.fbRecipe.SetTextIn (stIN := sttmpSkladnik, eLocation := E_BaseLocation.de, wsDescription := "Nazwa skladnika 1 DE");
	GVL.fbRecipe.SetMaxIn (stIN := sttmpSkladnik, rMax := 10000);
	GVL.fbRecipe.SetMinIn (stIN := sttmpSkladnik, rMin := 1);
	GVL.fbRecipe.SetValueIn (stIN := sttmpSkladnik, rValue := 1111);
	GVL.fbRecipe.SetDefaultValueIn (stIN := sttmpSkladnik, rDefaultValue := 1111);
	GVL.fbRecipe.SetUnitIn (stIN := sttmpSkladnik, sUnit := 'mm');
	bResult	:= GVL.fbRecipe.AddIngredientToTemplate (uiNumber := 1, stIngredient := sttmpSkladnik);
//test dodania
	AssertTrue (Condition := bResult, 																											Message := 'Test 06 - Blad utworzenia szablonu');
	AssertEquals_UINT (Expected := 1, Actual := GVL.fbRecipe.GetNumberIngredientOFTemplate (uiNumber := 1),										Message := 'Test 06a - Blad ilosci dodanych skladnikow');
	AssertEquals_WSTRING (Expected := "Nazwa skladnika 1 PL", Actual := GVL.fbRecipe.arrTemplates [1].arrIngredient [1].stTexts.arrText [1],	Message := 'Test 06b - bledna etykieta');
	AssertEquals_REAL (Expected := 1111, Actual := GVL.fbRecipe.arrTemplates [1].arrIngredient [1].rValue,										Message := 'Test 06c - bledna wartosc', Delta := 0);
	AssertEquals_REAL (Expected := 1111, Actual := GVL.fbRecipe.arrTemplates [1].arrIngredient [1].rDefaultValue,								Message := 'Test 06d - bledna wartosc domyslna', Delta := 0);
	AssertEquals_REAL (Expected := 1, Actual := GVL.fbRecipe.arrTemplates [1].arrIngredient [1].rMin,		 									Message := 'Test 06e - bledna wartosc min', Delta := 0);
	AssertEquals_REAL (Expected := 10000, Actual := GVL.fbRecipe.arrTemplates [1].arrIngredient [1].rMAX,		 								Message := 'Test 06f - bledna wartosc max', Delta := 0);
	AssertEquals_WSTRING (Expected := "mm", Actual := TO_WSTRING (GVL.fbRecipe.arrTemplates [1].arrIngredient [1].sUnit),		 				Message := 'Test 06g - bledna jednostka');

	GVL.fbRecipe.SetTextIn (stIN := sttmpSkladnik, eLocation := E_BaseLocation.pl, wsDescription := "Nazwa skladnika 2 PL");
	GVL.fbRecipe.SetTextIn (stIN := sttmpSkladnik, eLocation := E_BaseLocation.en, wsDescription := "Nazwa skladnika 2 EN");
	GVL.fbRecipe.SetTextIn (stIN := sttmpSkladnik, eLocation := E_BaseLocation.de, wsDescription := "Nazwa skladnika 2 DE");
	GVL.fbRecipe.SetMaxIn (stIN := sttmpSkladnik, rMax := 10000);
	GVL.fbRecipe.SetMinIn (stIN := sttmpSkladnik, rMin := 1);
	GVL.fbRecipe.SetValueIn (stIN := sttmpSkladnik, rValue := 1112);
	GVL.fbRecipe.SetDefaultValueIn (stIN := sttmpSkladnik, rDefaultValue := 1112);
	GVL.fbRecipe.SetUnitIn (stIN := sttmpSkladnik, sUnit := 'mm/s');
	bResult	:= GVL.fbRecipe.AddIngredientToTemplate (uiNumber := 1, stIngredient := sttmpSkladnik);
	
	AssertTrue (Condition := bResult, 																											Message := 'Test 07 - Blad utworzenia szablonu');
	AssertEquals_UINT (Expected := 2, Actual := GVL.fbRecipe.GetNumberIngredientOFTemplate (uiNumber := 1),										Message := 'Test 07a - Blad ilosci dodanych skladnikow');
	AssertEquals_WSTRING (Expected := "Nazwa skladnika 2 PL", Actual := GVL.fbRecipe.arrTemplates [1].arrIngredient [2].stTexts.arrText [1],	Message := 'Test 07b - bledna etykieta');
	AssertEquals_REAL (Expected := 1112, Actual := GVL.fbRecipe.arrTemplates [1].arrIngredient [2].rValue,										Message := 'Test 07c - bledna wartosc', Delta := 0);
	AssertEquals_REAL (Expected := 1112, Actual := GVL.fbRecipe.arrTemplates [1].arrIngredient [2].rDefaultValue,								Message := 'Test 07d - bledna wartosc domyslna', Delta := 0);
	AssertEquals_REAL (Expected := 1, Actual := GVL.fbRecipe.arrTemplates [1].arrIngredient [2].rMin,		 									Message := 'Test 07e - bledna wartosc min', Delta := 0);
	AssertEquals_REAL (Expected := 10000, Actual := GVL.fbRecipe.arrTemplates [1].arrIngredient [2].rMAX,		 								Message := 'Test 07f - bledna wartosc max', Delta := 0);
	AssertEquals_WSTRING (Expected := "mm/s", Actual := TO_WSTRING (GVL.fbRecipe.arrTemplates [1].arrIngredient [2].sUnit),		 			Message := 'Test 07g - bledna jednostka');

	GVL.fbRecipe.SetTextIn (stIN := sttmpSkladnik, eLocation := E_BaseLocation.pl, wsDescription := "Nazwa skladnika 3 PL");
	GVL.fbRecipe.SetTextIn (stIN := sttmpSkladnik, eLocation := E_BaseLocation.en, wsDescription := "Nazwa skladnika 3 EN");
	GVL.fbRecipe.SetTextIn (stIN := sttmpSkladnik, eLocation := E_BaseLocation.de, wsDescription := "Nazwa skladnika 3 DE");
	GVL.fbRecipe.SetMaxIn (stIN := sttmpSkladnik, rMax := 10000);
	GVL.fbRecipe.SetMinIn (stIN := sttmpSkladnik, rMin := 1);
	GVL.fbRecipe.SetValueIn (stIN := sttmpSkladnik, rValue := 1113);
	GVL.fbRecipe.SetDefaultValueIn (stIN := sttmpSkladnik, rDefaultValue := 1113);
	GVL.fbRecipe.SetUnitIn (stIN := sttmpSkladnik, sUnit := 'ms');
	bResult	:= GVL.fbRecipe.AddIngredientToTemplate (uiNumber := 1, stIngredient := sttmpSkladnik);
	
	AssertTrue (Condition := bResult, 																											Message := 'Test 08 - Blad utworzenia szablonu');
	AssertEquals_UINT (Expected := 3, Actual := GVL.fbRecipe.GetNumberIngredientOFTemplate (uiNumber := 1),										Message := 'Test 08a - Blad ilosci dodanych skladnikow');
	AssertEquals_WSTRING (Expected := "Nazwa skladnika 3 PL", Actual := GVL.fbRecipe.arrTemplates [1].arrIngredient [3].stTexts.arrText [1],	Message := 'Test 08b - bledna etykieta');
	AssertEquals_REAL (Expected := 1113, Actual := GVL.fbRecipe.arrTemplates [1].arrIngredient [3].rValue,										Message := 'Test 08c - bledna wartosc', Delta := 0);
	AssertEquals_REAL (Expected := 1113, Actual := GVL.fbRecipe.arrTemplates [1].arrIngredient [3].rDefaultValue,								Message := 'Test 08d - bledna wartosc domyslna', Delta := 0);
	AssertEquals_REAL (Expected := 1, Actual := GVL.fbRecipe.arrTemplates [1].arrIngredient [3].rMin,		 									Message := 'Test 08e - bledna wartosc min', Delta := 0);
	AssertEquals_REAL (Expected := 10000, Actual := GVL.fbRecipe.arrTemplates [1].arrIngredient [3].rMAX,		 								Message := 'Test 08f - bledna wartosc max', Delta := 0);
	AssertEquals_WSTRING (Expected := "ms", Actual := TO_WSTRING (GVL.fbRecipe.arrTemplates [1].arrIngredient [3].sUnit),		 				Message := 'Test 08g - bledna jednostka');

//Kolejny szablon
	GVL.fbRecipe.SetText (eLocation := E_BaseLocation.pl, wsDescription := "Nazwa szablonu 2 PL");
	GVL.fbRecipe.SetText (eLocation := E_BaseLocation.en, wsDescription := "Nazwa szablonu 2 EN");
	GVL.fbRecipe.SetText (eLocation := E_BaseLocation.de, wsDescription := "Nazwa szablonu 2 DE");
	bResult	:= GVL.fbRecipe.AddTemplates (stTexts	:= GVL.fbRecipe.GetTexts ());
	AssertTrue (Condition := bResult, 															Message := 'T09 - Blad utworzenia szablonu');
	AssertEquals_UINT (Expected := 2, Actual := GVL.fbRecipe.GetNumberOfTemplate (),			Message := 'T10 - Blad ilosci dodanych szablonow');
//skladnik
	GVL.fbRecipe.SetTextIn (stIN := sttmpSkladnik, eLocation := E_BaseLocation.pl, wsDescription := "Nazwa skladnika 1 PL");
	GVL.fbRecipe.SetTextIn (stIN := sttmpSkladnik, eLocation := E_BaseLocation.en, wsDescription := "Nazwa skladnika 1 EN");
	GVL.fbRecipe.SetTextIn (stIN := sttmpSkladnik, eLocation := E_BaseLocation.de, wsDescription := "Nazwa skladnika 1 DE");
	GVL.fbRecipe.SetMaxIn (stIN := sttmpSkladnik, rMax := 10000);
	GVL.fbRecipe.SetMinIn (stIN := sttmpSkladnik, rMin := 1);
	GVL.fbRecipe.SetValueIn (stIN := sttmpSkladnik, rValue := 1111);
	GVL.fbRecipe.SetDefaultValueIn (stIN := sttmpSkladnik, rDefaultValue := 1111);
	GVL.fbRecipe.SetUnitIn (stIN := sttmpSkladnik, sUnit := 'mm');
	bResult	:= GVL.fbRecipe.AddIngredientToTemplate (uiNumber := 2, stIngredient := sttmpSkladnik);

	AssertTrue (Condition := bResult, 																											Message := 'Test 11 - Blad utworzenia szablonu');
	AssertEquals_UINT (Expected := 1, Actual := GVL.fbRecipe.GetNumberIngredientOFTemplate (uiNumber := 2),										Message := 'Test 11a - Blad ilosci dodanych skladnikow');
	AssertEquals_WSTRING (Expected := "Nazwa skladnika 1 PL", Actual := GVL.fbRecipe.arrTemplates [2].arrIngredient [1].stTexts.arrText [1],	Message := 'Test 11b - bledna etykieta');
	AssertEquals_REAL (Expected := 1111, Actual := GVL.fbRecipe.arrTemplates [2].arrIngredient [1].rValue,										Message := 'Test 11c - bledna wartosc', Delta := 0);
	AssertEquals_REAL (Expected := 1111, Actual := GVL.fbRecipe.arrTemplates [2].arrIngredient [1].rDefaultValue,								Message := 'Test 11d - bledna wartosc domyslna', Delta := 0);
	AssertEquals_REAL (Expected := 1, Actual := GVL.fbRecipe.arrTemplates [2].arrIngredient [1].rMin,		 									Message := 'Test 11e - bledna wartosc min', Delta := 0);
	AssertEquals_REAL (Expected := 10000, Actual := GVL.fbRecipe.arrTemplates [2].arrIngredient [1].rMAX,		 								Message := 'Test 11f - bledna wartosc max', Delta := 0);
	AssertEquals_WSTRING (Expected := "mm", Actual := TO_WSTRING (GVL.fbRecipe.arrTemplates [2].arrIngredient [1].sUnit),		 				Message := 'Test 11g - bledna jednostka');
*)
END_METHOD

METHOD PROTECTED T22_TestAddRecipeFromTemplate
VAR
	bResult: BOOL;
	sttmpLabel: ST_BaseLabel;
END_VAR
IF (TcUnit.TEST_ORDERED ('T22_TestAddRecipeFromTemplate')) THEN
	MEMSET (
		destAddr		:= ADR (GVL.fbRecipe.arrRecipes),
		fillByte		:= 0,
		n				:= SIZEOF (GVL.fbRecipe.arrRecipes)
	);
	WRITE_PROTECTED_UINT (ADR(GVL.fbRecipe.uiNumberOfRecipes), 0);

	
	GVL.fbRecipe.SetText (eLocation := E_BaseLocation.pl, wsDescription := "Nazwa receptury PL");
	GVL.fbRecipe.SetText (eLocation := E_BaseLocation.en, wsDescription := "Nazwa receptury EN");
	GVL.fbRecipe.SetText (eLocation := E_BaseLocation.de, wsDescription := "Nazwa receptury DE");
	

	bResult		:= GVL.fbRecipe.AddRecipeFromTemplate (uiNumberTemplates := 1, stTexts := GVL.fbRecipe.GetTexts ());	

	AssertTrue (Condition := bResult, Message := 'Test 01 - Blad utworzenia receptury');
	AssertEquals_UINT (Expected := 1, Actual := GVL.fbRecipe.GetNumberOfRecipe (), Message := 'Test 02 - Blad ilosci dodanych receptur');
	
	sttmpLabel 			:= GVL.fbRecipe.GetNamesOfRecipe (uiNumber := 1);
	AssertEquals_WSTRING (Expected := "Nazwa receptury PL", Actual := sttmpLabel.arrText [E_BaseLocation.pl], Message := 'Test 03 - bledna nazwa receptury');

	AssertEquals_UINT (Expected := 3, Actual := GVL.fbRecipe.GetNumberIngredientOfRecipe (uiNumer := 1), Message := 'Test 04 - Blad ilosci dodanych skladnikow');
	AssertEquals_WSTRING (Expected := "Nazwa skladnika 1 PL", Actual := GVL.fbRecipe.arrRecipes [1].arrIngredient [1].stTexts.arrText [1],	Message := 'Test 05 - bledna etykieta');
	AssertEquals_REAL (Expected := 1111, Actual := GVL.fbRecipe.arrRecipes [1].arrIngredient [1].rValue, 						Message := 'Test 06 - bledna wartosc', Delta := 0);
	AssertEquals_REAL (Expected := 1111, Actual := GVL.fbRecipe.arrRecipes [1].arrIngredient [1].rDefaultValue, 				Message := 'Test 07 - bledna wartosc domyslna', Delta := 0);
	AssertEquals_REAL (Expected := 1, Actual := GVL.fbRecipe.arrRecipes [1].arrIngredient [1].rMin, 							Message := 'Test 08 - bledna wartosc min', Delta := 0);
	AssertEquals_REAL (Expected := 10000, Actual := GVL.fbRecipe.arrRecipes [1].arrIngredient [1].rMax, 						Message := 'Test 09 - bledna wartosc max', Delta := 0);
	AssertEquals_WSTRING (Expected := "mm", Actual := TO_WSTRING (GVL.fbRecipe.arrRecipes [1].arrIngredient [1].sUnit), 		Message := 'Test 10 - bledna jednostka');

	TcUnit.TEST_FINISHED ();

END_IF
END_METHOD

METHOD PUBLIC T23_TestDeleteRecipe
VAR
	bresult			: BOOL;
	sttmpLabel: ST_BaseLabel;
END_VAR
IF (TcUnit.TEST_ORDERED ('T23_TestDeleteRecipe')) THEN
	bresult	:= GVL.fbRecipe.DeleteRecipe (uiNumber	:= 1);
	AssertTrue (Condition := bresult, Message := 'Test 01 - Bladna wynik usuwania receptury');
	AssertEquals_UINT (Expected := 0, Actual := GVL.fbRecipe.GetNumberOfRecipe (), Message := 'Test 02 - bledna ilosc receptur');

	GVL.fbRecipe.SetText (eLocation := E_BaseLocation.pl, wsDescription := "Nazwa receptury 1 PL");
	GVL.fbRecipe.SetText (eLocation := E_BaseLocation.en, wsDescription := "Nazwa receptury 1 EN");
	GVL.fbRecipe.SetText (eLocation := E_BaseLocation.de, wsDescription := "Nazwa receptury 1 DE");
	bresult := GVL.fbRecipe.AddRecipeFromTemplate (uiNumberTemplates := 1, stTexts := GVL.fbRecipe.GetTexts ());
	AssertTrue (Condition := bresult, Message := 'Test 03a - Blad dodania receptury');
	AssertEquals_UINT (Expected := 1, Actual := GVL.fbRecipe.GetNumberOfRecipe (), Message := 'Test 20a - bledna ilosc receptur');
	
	GVL.fbRecipe.SetText (eLocation := E_BaseLocation.pl, wsDescription := "Nazwa receptury 2 PL");
	GVL.fbRecipe.SetText (eLocation := E_BaseLocation.en, wsDescription := "Nazwa receptury 2 EN");
	GVL.fbRecipe.SetText (eLocation := E_BaseLocation.de, wsDescription := "Nazwa receptury 2 DE");
	bresult := GVL.fbRecipe.AddRecipeFromTemplate (uiNumberTemplates := 1, stTexts := GVL.fbRecipe.GetTexts ());
	AssertTrue (Condition := bresult, Message := 'Test 03b - Blad dodania receptury');
	AssertEquals_UINT (Expected := 2, Actual := GVL.fbRecipe.GetNumberOfRecipe (), Message := 'Test 20b - bledna ilosc receptur');

	GVL.fbRecipe.SetText (eLocation := E_BaseLocation.pl, wsDescription := "Nazwa receptury 3 PL");
	GVL.fbRecipe.SetText (eLocation := E_BaseLocation.en, wsDescription := "Nazwa receptury 3 EN");
	GVL.fbRecipe.SetText (eLocation := E_BaseLocation.de, wsDescription := "Nazwa receptury 3 DE");
	bresult := GVL.fbRecipe.AddRecipeFromTemplate (uiNumberTemplates := 1, stTexts := GVL.fbRecipe.GetTexts ());
	AssertTrue (Condition := bresult, Message := 'Test 03c - Blad dodania receptury');
	AssertEquals_UINT (Expected := 3, Actual := GVL.fbRecipe.GetNumberOfRecipe (), Message := 'Test 20c - bledna ilosc receptur');

	GVL.fbRecipe.SetText (eLocation := E_BaseLocation.pl, wsDescription := "Nazwa receptury 4 PL");
	GVL.fbRecipe.SetText (eLocation := E_BaseLocation.en, wsDescription := "Nazwa receptury 4 EN");
	GVL.fbRecipe.SetText (eLocation := E_BaseLocation.de, wsDescription := "Nazwa receptury 4 DE");
	bresult := GVL.fbRecipe.AddRecipeFromTemplate (uiNumberTemplates := 1, stTexts := GVL.fbRecipe.GetTexts ());
	AssertTrue (Condition := bresult, Message := 'Test 03d - Blad dodania receptury');
	AssertEquals_UINT (Expected := 4, Actual := GVL.fbRecipe.GetNumberOfRecipe (), Message := 'Test 20d - bledna ilosc receptur');

	bresult	:= GVL.fbRecipe.DeleteRecipe (uiNumber	:= 2);
	AssertTrue (Condition := bresult, Message := 'Test 07 - Bladna wynik usuwania receptury');
	AssertEquals_UINT (Expected := 3, Actual := GVL.fbRecipe.GetNumberOfRecipe (), Message := 'Test 08 - bledna ilosc receptur');

	sttmpLabel 			:= GVL.fbRecipe.GetNamesOfRecipe (uiNumber := 2);
	AssertEquals_WSTRING (Expected := "Nazwa receptury 3 PL", Actual := sttmpLabel.arrText [E_BaseLocation.pl], Message := 'Test 09a - bledna nazwa receptury');
	sttmpLabel 			:= GVL.fbRecipe.GetNamesOfRecipe (uiNumber := 3);
	AssertEquals_WSTRING (Expected := "Nazwa receptury 4 PL", Actual := sttmpLabel.arrText [E_BaseLocation.pl], Message := 'Test 09b - bledna nazwa receptury');
	
	TcUnit.TEST_FINISHED ();
END_IF
END_METHOD

METHOD PROTECTED T24_TestCopyRecipeToNewRecipe
VAR
	bresult		: BOOL;
	sttmpLabel: ST_BaseLabel;
END_VAR
IF (TcUnit.TEST_ORDERED ('T24_TestCopyRecipeToNewRecipe')) THEN
	GVL.fbRecipe.SetText (eLocation := E_BaseLocation.pl, wsDescription	:= "Nazwa receptury klon PL");
	GVL.fbRecipe.SetText (eLocation := E_BaseLocation.en, wsDescription	:= "Nazwa receptury klon EN");
	GVL.fbRecipe.SetText (eLocation := E_BaseLocation.de, wsDescription	:= "Nazwa receptury klon DE");
	

	bresult		:= GVL.fbRecipe.AddRecipeFromRecipe (uiNumberRecipe := 1, stTexts := GVL.fbRecipe.GetTexts ());	

	AssertTrue (Condition := bresult, Message := 'Test 01 - Blad utworzenia receptury');
	AssertEquals_UINT (Expected := 4, Actual := GVL.fbRecipe.GetNumberOfRecipe (), Message := 'Test 02 - Blad ilosci dodanych receptur');
	sttmpLabel 			:= GVL.fbRecipe.GetNamesOfRecipe (uiNumber := 4);
	AssertEquals_WSTRING (Expected := "Nazwa receptury klon PL", Actual := sttmpLabel.arrText [E_BaseLocation.pl], Message := 'Test 03 - bledna nazwa receptury');

	AssertEquals_UINT (Expected := 3, Actual := GVL.fbRecipe.GetNumberIngredientOfRecipe (uiNumer := 1), Message := 'Test 04 - Blad ilosci dodanych skladnikow');
	AssertEquals_WSTRING (Expected := "Nazwa skladnika 1 PL", Actual := GVL.fbRecipe.arrRecipes [4].arrIngredient [1].stTexts.arrText [1], 	Message := 'Test 05 - bledna etykieta');
	AssertEquals_REAL (Expected := 1111, Actual := GVL.fbRecipe.arrRecipes [4].arrIngredient [1].rValue, 							Message := 'Test 06 - bledna wartosc', Delta := 0);
	AssertEquals_REAL (Expected := 1111, Actual := GVL.fbRecipe.arrRecipes [4].arrIngredient [1].rDefaultValue, 					Message := 'Test 07 - bledna wartosc domyslna', Delta := 0);
	AssertEquals_REAL (Expected := 1, Actual := GVL.fbRecipe.arrRecipes [4].arrIngredient [1].rMIN, 								Message := 'Test 08 - bledna wartosc min', Delta := 0);
	AssertEquals_REAL (Expected := 10000, Actual := GVL.fbRecipe.arrRecipes [4].arrIngredient [1].rMAX, 							Message := 'Test 09 - bledna wartosc max', Delta := 0);
	AssertEquals_WSTRING (Expected := "mm", Actual := TO_WSTRING (GVL.fbRecipe.arrRecipes [4].arrIngredient [1].sUnit),			Message := 'Test 10 - bledna jednostka');

	
	TcUnit.TEST_FINISHED ();
END_IF
END_METHOD

METHOD INTERNAL T99_Test
VAR_INST
	bFinish	: BOOL;
	bT99Test: BOOL;
END_VAR
IF (TcUnit.TEST_ORDERED ('T99_Test')) THEN
	bT99Test			:= TRUE;

	GVL_Variable.fbPB1.ExecuteEveryCycle_Test ();
	GVL_Variable.fbPB1.ExecuteEveryCycle_Operation ();
	GVL_Variable.fbPB1.ExecuteEveryCycle_Status ();
	GVL_Variable.fbPB1.ExecuteEveryCycle_Error ();
	
	IF bFinish THEN
		bT99Test		:= FALSE;
		TcUnit.TEST_FINISHED ();
	END_IF
END_IF
END_METHOD

END_FUNCTION_BLOCK

// ---- TESTs/PRG_Test.TcPOU
PROGRAM PRG_Test
VAR
	fbBaseTimeTest			: FB_BaseTimeTest;
	fbCommandTest			: FB_CommandTest;
	fbImpulsTest			: FB_Impulstest;

	fbItemTest				: FB_ItemTest;
//	fbBaseTest				: FB_Basetest;
//	fbComponentTest			: FB_ElementTest;
//
//	fbLoggerTest			: FB_LoggerTest;

END_VAR


	TcUnit.RUN_IN_SEQUENCE ();

END_PROGRAM
